(* IEC 61131-3 sources: eCockpitGit/test_project/src/%F%00 Library/%F%Common Functions/%F%Dynamic Array/%POU%FB_DynamicArray, 7 files *)

(* ---- %METH%allocate.st ---- *)
//NON-Blocking method, is not threadsafe without calling getExclusive access before use
//Pre-allocates a given size to the array
// |**Version**|**Author**| **Date** |**Changes**
// | 1         | NSN      | 03-03-22 | Creation
METHOD allocate :SLMResult
VAR_INPUT
	size			:WORD;		//Size to allocate to array
END_VAR
VAR
	newByteSize		:DWORD;
	newArrayBuffer	:POINTER TO ARRAY[0..99] OF BYTE;
END_VAR
(*%!%__DELIMITER__%!%*)
IF size > S_blockSize THEN
	//Size is corrected to increment size
	size							:=		(((size - 1) / S_increment) + 1) * S_increment;
	//Byte size is calculated
	newByteSize						:=		size * S_elementSize;
	newArrayBuffer					:=		__NEW(BYTE,newByteSize);
	//If the memory manager fails, the registerering fails
	IF newArrayBuffer = 0 THEN
		allocate.success	:=		FALSE;
		allocate.code		:=		ERCodes.FB_DynamicArray_allocateInternal;
		allocate.reason		:=		GTErrors.EoutOfDynamicMemory;
		RETURN;
	END_IF
	//The contens of the old buffer is copied to the new buffer
	IF S_lenght > 0 THEN
		SysMem.SysMemCpy(pDest:=newArrayBuffer,pSrc:=S_array^,udiCount:=S_lenght * S_elementSize);
	END_IF
	//Old array memory is deleted, and new one is use
	FU_SafeDelete(pMem:=S_array^);
	S_array^						:=		newArrayBuffer;
	S_blockSize						:=		size;
END_IF

(* ---- %METH%appendElement.st ---- *)
//NON-Blocking method, is not threadsafe without calling getExclusive access before use
//Appends element to array
// |**Version**|**Author**| **Date** |**Changes**
// | 1         | NSN      | 03-03-22 | Creation
METHOD appendElement : SLMResult
VAR_INPUT
	element			:POINTER TO BYTE;	//Element to check
	elementSize		:WORD;		//Size of element
END_VAR
VAR_OUTPUT
	index			:WORD;
END_VAR

(*%!%__DELIMITER__%!%*)
IF S_lenght < S_maxSize THEN
	IF S_map THEN
		IF checkExists(element:=element,elementSize:=elementSize) THEN
			appendElement.success		:=		FALSE;
			appendElement.code			:=		ERCodes.FB_DynamicArray_addElement;
			appendElement.reason		:=		GTErrors.EelementInArray;
			RETURN;
		END_IF
	END_IF
	//If array is full, then more space is allocated
	IF S_lenght = S_blockSize THEN
		appendElement					:=		allocate(size:=S_blockSize + 1);
		IF NOT(appendElement.success) THEN
			RETURN;
		END_IF
	END_IF

	SysMem.SysMemCpy(pDest:=S_array^ + (S_lenght * S_elementSize),pSrc:=element,udiCount:=MIN(elementSize,S_elementSize));
	index										:=		S_lenght;
	S_lenght									:=		S_lenght + 1;
ELSE
	appendElement.success				:=		FALSE;
	appendElement.code					:=		ERCodes.FB_DynamicArray_addElement;
	appendElement.reason				:=		GTErrors.EarrayFull;
END_IF

(* ---- %METH%checkAgainst.st ---- *)
//BLOCKING Method, method will block thread until exclusive access to array is available
//Compares the given element to the element on the index in the array
//Returns true if element is the same
// |**Version**|**Author**| **Date** |**Changes**
// | 1         | NSN      | 03-03-22 | Creation
METHOD checkAgainst : BOOL
VAR_INPUT
	element		:POINTER TO BYTE;	//Element to check
	elementSize	:WORD;		//Size of element
	index		:WORD;		//Index
END_VAR
VAR
	i			:WORD;
END_VAR
(*%!%__DELIMITER__%!%*)
IF index < S_lenght THEN
	checkAgainst		:=		compare(elementInt:=S_array^ + (index * S_elementSize),elementExt:=element,elementExtSize:=elementSize);
END_IF

(* ---- %METH%checkExists.st ---- *)
//NON-Blocking method, is not threadsafe without calling getExclusive access before use
//Checks if element exist in array, and returns index of element in array
//Returns true if element is found
// |**Version**|**Author**| **Date** |**Changes**
// | 1         | NSN      | 03-03-22 | Creation
METHOD checkExists : BOOL
VAR_INPUT
	element		:POINTER TO BYTE;	//Element to check
	elementSize	:WORD;		//Size of element
END_VAR
VAR_OUTPUT
	index		:WORD;		//Index of found element
END_VAR
(*%!%__DELIMITER__%!%*)
IF S_lenght > 0 THEN
	//Array is searched until element is found
	FOR index := 0 TO S_lenght - 1 DO
		IF compare(elementInt:=S_array^ + (index * S_elementSize),elementExt:=element,elementExtSize:=elementSize) THEN
			checkExists		:=		TRUE;
			RETURN;
		END_IF
	END_FOR
END_IF
index								:=		0;

(* ---- %METH%getElementByIndex.st ---- *)
//NON-Blocking method, is not threadsafe without calling getExclusive access before use
//Copies data from index in array to given memory position
// |**Version**|**Author**| **Date** |**Changes**
// | 1         | NSN      | 07-03-22 | Creation
METHOD getElementByIndex : SLMResult
VAR_INPUT
	element			:POINTER TO BYTE;
	elementSize		:WORD;
	index			:WORD;
END_VAR

(*%!%__DELIMITER__%!%*)
IF index < S_lenght THEN
	SysMem.SysMemCpy(pDest:=element,pSrc:=S_array^ + (index * S_elementSize),udiCount:=MIN(S_elementSize,elementSize));
ELSE
	getElementByIndex.success		:=		FALSE;
	getElementByIndex.code			:=		ERCodes.FB_DynamicArray_removeElementByIndex;
	getElementByIndex.reason		:=		GTErrors.EindexOutOfRange;
END_IF

(* ---- %METH%removeElement.st ---- *)
//NON-Blocking method, is not threadsafe without calling getExclusive access before use
//Finds and removes the given element from the array, if multiple are found the amount of elements removed are limited by the amount given
// |**Version**|**Author**| **Date** |**Changes**
// | 1         | NSN      | 07-03-22 | Creation
METHOD removeElement
VAR_INPUT
	element			:POINTER TO BYTE;	//Element to remove
	elementSize		:WORD;		//Size of element
	amount			:WORD;		//Max amount of same elements to remove from array, 0 means all
END_VAR
VAR
	i				:WORD;
	offset			:WORD;
END_VAR
(*%!%__DELIMITER__%!%*)
IF S_lenght > 0 THEN
	FOR i := 0 TO S_lenght - 1 DO
		IF compare(elementInt:=S_array^ + (i * S_elementSize),elementExt:=element,elementExtSize:=elementSize) AND (offset < amount OR amount = 0) THEN
			offset				:=		offset + 1;
		ELSIF offset > 0 THEN
			SysMem.SysMemCpy(pDest:=S_array^ + ((i - offset) * S_elementSize),pSrc:=S_array^ + (i * S_elementSize),udiCount:=S_elementSize);
		END_IF
	END_FOR
	S_lenght						:=		S_lenght - offset;
	IF S_lenght = 0 THEN
		S_blockSize					:=		0;
		FU_SafeDelete(pMem:=S_array^);
	END_IF
END_IF

(* ---- %METH%removeElementByIndex.st ---- *)
//NON-Blocking method, is not threadsafe without calling getExclusive access before use
//Removes a given index from the array, by shifting all memory after it over it
// |**Version**|**Author**| **Date** |**Changes**
// | 1         | NSN      | 07-03-22 | Creation
METHOD removeElementByIndex : SLMResult
VAR_INPUT
	index			:WORD;		//Index to remove element from
END_VAR

(*%!%__DELIMITER__%!%*)
IF index < S_lenght THEN
	S_lenght									:=		S_lenght - 1;
	SysMem.SysMemCpy(pDest:=S_array^ + (index * S_elementSize),pSrc:=S_array^ + ((index + 1) * S_elementSize),udiCount:=(S_lenght - index) * S_elementSize);
	IF S_lenght = 0 THEN
		S_blockSize								:=		0;
		FU_SafeDelete(pMem:=S_array^);
	END_IF
ELSE
	removeElementByIndex.success		:=		FALSE;
	removeElementByIndex.code			:=		ERCodes.FB_DynamicArray_removeElementByIndex;
	removeElementByIndex.reason			:=		GTErrors.EindexOutOfRange;
END_IF
